KUKA KRL program: dai_chg_GRH_01.src, dai_chg_GRH_01.dat

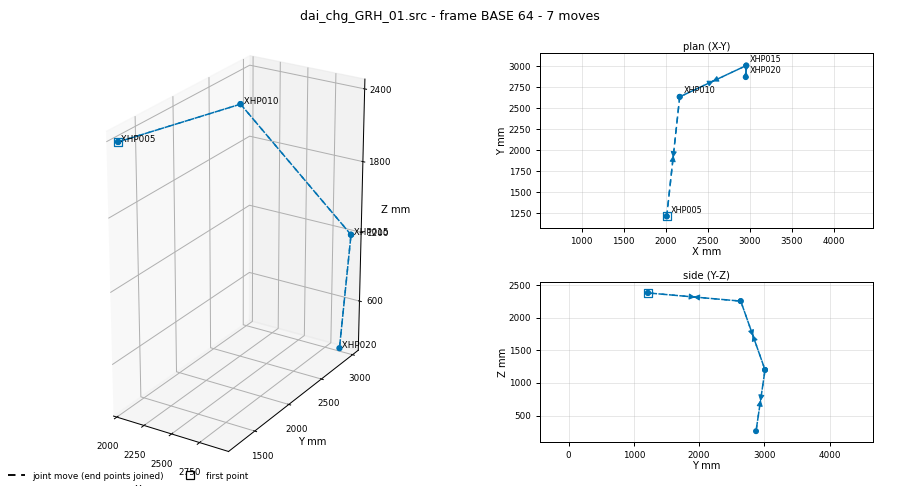
[picture p0: tool path of dai_chg_GRH_01.src in frame BASE 64, 7 of 9 moves have a stored position in this frame; points joined in program order, loops and branches not executed]
--- dai_chg_GRH_01.src ---
&ACCESS RVP
&REL 21
&COMMENT dai_chg_060GRH101
&USER PKL_AST
&PARAM version = 0.1
&PARAM DISKPATH = KRC:\R1\H_Prog
DEF dai_chg_GRH_01( )
;FOLD INI
  ;FOLD BASISTECH INI
    GLOBAL INTERRUPT DECL 3 WHEN $STOPMESS==TRUE DO IR_STOPM ( )
    BAS (#INITMOV,0 )
  ;ENDFOLD (BASISTECH INI)
;FOLD USER INI

;Make your modifications here
;FOLD COLLISION_V_3.01 INI ;%{E}
    IF (COLLISION_DATA[1].I_NR>0) THEN
    GLOBAL INTERRUPT DECL 21 WHEN $IN[COLLISION_DATA[1].I_NR]==FALSE DO COLLSTOP (1,0 )
    ENDIF
    IF (COLLISION_DATA[2].I_NR>0) THEN
    GLOBAL INTERRUPT DECL 22 WHEN $IN[COLLISION_DATA[2].I_NR]==FALSE DO COLLSTOP (2,0 )
    ENDIF
    IF (COLLISION_DATA[3].I_NR>0) THEN
    GLOBAL INTERRUPT DECL 23 WHEN $IN[COLLISION_DATA[3].I_NR]==FALSE DO COLLSTOP (3,0 )
    ENDIF
    IF (COLLISION_DATA[4].I_NR>0) THEN
    GLOBAL INTERRUPT DECL 24 WHEN $IN[COLLISION_DATA[4].I_NR]==FALSE DO COLLSTOP (4,0 )
    ENDIF
;ENDFOLD (Collision)

;ENDFOLD (USER INI)

;ENDFOLD (INI)
;FOLD ; Anlagenbezeichn: HC53_C    Stations-Nr: 060RB_100;%{PE}
;FOLD Parameters ;%{h}
;Params IlfProvider=kukaroboter.basistech.inlineforms.comments.comment; Kuka.Content=Anlagenbezeichn: HC53_C    Stations-Nr: 060RB_100
;ENDFOLD
;ENDFOLD
;FOLD ; Stand / Version: V1.0;%{PE}
;FOLD Parameters ;%{h}
;Params IlfProvider=kukaroboter.basistech.inlineforms.comments.comment; Kuka.Content=Stand / Version: V1.0
;ENDFOLD
;ENDFOLD
;FOLD ; Name Bearbeiter: EBZ-AE;%{PE}
;FOLD Parameters ;%{h}
;Params IlfProvider=kukaroboter.basistech.inlineforms.comments.comment; Kuka.Content=Name Bearbeiter: EBZ-AE
;ENDFOLD
;ENDFOLD
;FOLD ; Translator Version:29.01.2024 - Version 15.08;%{PE}
;FOLD Parameters ;%{h}
;Params IlfProvider=kukaroboter.basistech.inlineforms.comments.comment; Kuka.Content=Translator Version:29.01.2024 - Version 15.08
;ENDFOLD
;ENDFOLD


;FOLD ; This program has been cleaned by KANERT_Makro. High risk of crash!!! Check the program carefully before deleting this comment. ;%{PE}
;FOLD Parameters ;%{h}
;Params IlfProvider=kukaroboter.basistech.inlineforms.comments.comment; Kuka.Content=This program has been cleaned by KANERT_Makro. High risk of crash!!! Check the program carefully before deleting this comment.
;ENDFOLD
WAIT FOR FALSE
;ENDFOLD
REPEAT
;fold MSG_T1
MSG_SHOW("DAI_H_Prog",#quit,999,"dai_toolchange_0")
;endfold
; ***************************************
; A T T E N T I O N !!! Only drive in $T1
; A C H T U N G !!! Nur in $T1 abfahren
; ***************************************
UNTIL $T1 == TRUE
;FOLD PTP HOME Vel=100 % DEFAULT ;%{PE}
;FOLD Parameters ;%{h}
;Params IlfProvider=kukaroboter.basistech.inlineforms.movement.old; Kuka.IsGlobalPoint=False; Kuka.PointName=HOME; Kuka.BlendingEnabled=False; Kuka.MoveDataPtpName=DEFAULT; Kuka.VelocityPtp=100; Kuka.CurrentCDSetIndex=0; Kuka.MovementParameterFieldEnabled=True; IlfCommand=PTP
;ENDFOLD
$BWDSTART = FALSE
PDAT_ACT = PDEFAULT
FDAT_ACT = FHOME
BAS(#PTP_PARAMS, 100.0)
SET_CD_PARAMS (0)
PTP XHOME
;ENDFOLD

;Dynamische Pruefung Teil vorhanden
;FOLD PartPresent.CheckOff #1:5277, #2:5278, #3:1025, #4:1025, #5:1025, #6:1025, Bounce Time:100, Constant: Yes;%{PE}%
CheckPartPresent(5277,5278,1025,1025,1025,1025,100, True,FALSE)
;ENDFOLD
;FOLD DAI_GripValve.Valve2 State: Fixierstift Ausfahren Gs, Check: No, 060GRH101-QM1 ;%{PE}
ActuateValve(2,1, FALSE ,FALSE)
;ENDFOLD
;FOLD DAI_GripValve.Valve3 State: Spanner Oeffnen Gs, Check: No, 060GRH101-QM2 ;%{PE}
ActuateValve(3,1, FALSE ,FALSE)
;ENDFOLD
;FOLD DAI_GripValve.Valve4 State: Spanner Oeffnen Gs, Check: No, 060GRH101-QM3 ;%{PE}
ActuateValve(4,1, FALSE ,FALSE)
;ENDFOLD

;Greifer-Ventile betatigen/pruefen
;FOLD DAI_GripValveCheck.Valve2 State:Fixierstift Ausfahren Gs, 060GRH101-QM1;%{PE}%
CheckValveState(2,1)
;ENDFOLD
;FOLD DAI_GripValveCheck.Valve3 State:Spanner Oeffnen Gs, 060GRH101-QM2;%{PE}%
CheckValveState(3,1)
;ENDFOLD
;FOLD DAI_GripValveCheck.Valve4 State:Spanner Oeffnen Gs, 060GRH101-QM3;%{PE}%
CheckValveState(4,1)
;ENDFOLD

; Weg zu Ablageposition teachen
; Teach PTP-Way to depositing-position
;FOLD PTP HP005 Vel=100 % PDAT1 Tool[64]:Zero Base[64]:Zero ;%{PE}
;FOLD Parameters ;%{h}
;Params IlfProvider=kukaroboter.basistech.inlineforms.movement.old; Kuka.IsGlobalPoint=False; Kuka.PointName=HP005; Kuka.BlendingEnabled=False; Kuka.MoveDataPtpName=PDAT1; Kuka.VelocityPtp=100; Kuka.CurrentCDSetIndex=0; Kuka.MovementParameterFieldEnabled=True; IlfCommand=PTP
;ENDFOLD
$BWDSTART = FALSE
PDAT_ACT = PPDAT1
FDAT_ACT = FHP005
BAS(#PTP_PARAMS, 100.0)
SET_CD_PARAMS (0)
PTP XHP005
;ENDFOLD
;FOLD PTP HP010 Vel=100 % PDAT2 Tool[64]:Zero Base[64]:Zero ;%{PE}
;FOLD Parameters ;%{h}
;Params IlfProvider=kukaroboter.basistech.inlineforms.movement.old; Kuka.IsGlobalPoint=False; Kuka.PointName=HP010; Kuka.BlendingEnabled=False; Kuka.MoveDataPtpName=PDAT2; Kuka.VelocityPtp=100; Kuka.CurrentCDSetIndex=0; Kuka.MovementParameterFieldEnabled=True; IlfCommand=PTP
;ENDFOLD
$BWDSTART = FALSE
PDAT_ACT = PPDAT2
FDAT_ACT = FHP010
BAS(#PTP_PARAMS, 100.0)
SET_CD_PARAMS (0)
PTP XHP010
;ENDFOLD
;FOLD PTP HP015 Vel=100 % PDAT3 Tool[64]:Zero Base[64]:Zero ;%{PE}
;FOLD Parameters ;%{h}
;Params IlfProvider=kukaroboter.basistech.inlineforms.movement.old; Kuka.IsGlobalPoint=False; Kuka.PointName=HP015; Kuka.BlendingEnabled=False; Kuka.MoveDataPtpName=PDAT3; Kuka.VelocityPtp=100; Kuka.CurrentCDSetIndex=0; Kuka.MovementParameterFieldEnabled=True; IlfCommand=PTP
;ENDFOLD
$BWDSTART = FALSE
PDAT_ACT = PPDAT3
FDAT_ACT = FHP015
BAS(#PTP_PARAMS, 100.0)
SET_CD_PARAMS (0)
PTP XHP015
;ENDFOLD

; Ablageposition teachen
; depositing-position
;FOLD PTP HP020 Vel=100 % PDAT4 Tool[64]:Zero Base[64]:Zero ;%{PE}
;FOLD Parameters ;%{h}
;Params IlfProvider=kukaroboter.basistech.inlineforms.movement.old; Kuka.IsGlobalPoint=False; Kuka.PointName=HP020; Kuka.BlendingEnabled=False; Kuka.MoveDataPtpName=PDAT4; Kuka.VelocityPtp=100; Kuka.CurrentCDSetIndex=0; Kuka.MovementParameterFieldEnabled=True; IlfCommand=PTP
;ENDFOLD
$BWDSTART = FALSE
PDAT_ACT = PPDAT4
FDAT_ACT = FHP020
BAS(#PTP_PARAMS, 100.0)
SET_CD_PARAMS (0)
PTP XHP020
;ENDFOLD

;fold Ablageposition erreicht | depositing-position reeached
MSG_SHOW("DAI_H_Prog",#quit,999,"dai_toolchange_1")
;endfold
WAIT FOR  $IN[1026]==TRUE ;

REPEAT
;fold MSG_T1
MSG_SHOW("DAI_H_Prog",#quit,999,"dai_toolchange_0")
;endfold
; ***************************************
; A T T E N T I O N !!! Only drive in $T1
; A C H T U N G !!! Nur in $T1 abfahren
; ***************************************
UNTIL $T1 == TRUE

; Teache Weg zurueck zu Homeposition
; Teach PTP-way back to home
;FOLD PTP HP025 Vel=100 % PDAT5 Tool[64]:Zero Base[64]:Zero ;%{PE}
;FOLD Parameters ;%{h}
;Params IlfProvider=kukaroboter.basistech.inlineforms.movement.old; Kuka.IsGlobalPoint=False; Kuka.PointName=HP025; Kuka.BlendingEnabled=False; Kuka.MoveDataPtpName=PDAT5; Kuka.VelocityPtp=100; Kuka.CurrentCDSetIndex=0; Kuka.MovementParameterFieldEnabled=True; IlfCommand=PTP
;ENDFOLD
$BWDSTART = FALSE
PDAT_ACT = PPDAT5
FDAT_ACT = FHP025
BAS(#PTP_PARAMS, 100.0)
SET_CD_PARAMS (0)
PTP XHP025
;ENDFOLD
;FOLD PTP HP030 Vel=100 % PDAT6 Tool[64]:Zero Base[64]:Zero ;%{PE}
;FOLD Parameters ;%{h}
;Params IlfProvider=kukaroboter.basistech.inlineforms.movement.old; Kuka.IsGlobalPoint=False; Kuka.PointName=HP030; Kuka.BlendingEnabled=False; Kuka.MoveDataPtpName=PDAT6; Kuka.VelocityPtp=100; Kuka.CurrentCDSetIndex=0; Kuka.MovementParameterFieldEnabled=True; IlfCommand=PTP
;ENDFOLD
$BWDSTART = FALSE
PDAT_ACT = PPDAT6
FDAT_ACT = FHP030
BAS(#PTP_PARAMS, 100.0)
SET_CD_PARAMS (0)
PTP XHP030
;ENDFOLD
;FOLD PTP HP035 Vel=100 % PDAT7 Tool[64]:Zero Base[64]:Zero ;%{PE}
;FOLD Parameters ;%{h}
;Params IlfProvider=kukaroboter.basistech.inlineforms.movement.old; Kuka.IsGlobalPoint=False; Kuka.PointName=HP035; Kuka.BlendingEnabled=False; Kuka.MoveDataPtpName=PDAT7; Kuka.VelocityPtp=100; Kuka.CurrentCDSetIndex=0; Kuka.MovementParameterFieldEnabled=True; IlfCommand=PTP
;ENDFOLD
$BWDSTART = FALSE
PDAT_ACT = PPDAT7
FDAT_ACT = FHP035
BAS(#PTP_PARAMS, 100.0)
SET_CD_PARAMS (0)
PTP XHP035
;ENDFOLD

;FOLD PTP HOME Vel=100 % DEFAULT;%{PE}
;FOLD Parameters ;%{h}
;Params IlfProvider=kukaroboter.basistech.inlineforms.movement.old; Kuka.IsGlobalPoint=False; Kuka.PointName=HOME; Kuka.BlendingEnabled=False; Kuka.MoveDataPtpName=DEFAULT; Kuka.VelocityPtp=100; Kuka.CurrentCDSetIndex=0; Kuka.MovementParameterFieldEnabled=True; IlfCommand=PTP
;ENDFOLD
$BWDSTART = FALSE
PDAT_ACT = PDEFAULT
FDAT_ACT = FHOME
BAS(#PTP_PARAMS, 100.0)
SET_CD_PARAMS (0)
PTP XHOME
;ENDFOLD

END

--- dai_chg_GRH_01.dat ---
&ACCESS RVP
&REL 22
&COMMENT dai_chg_060GRH101
&USER PKL_AST
&PARAM version = 0.1
&PARAM DISKPATH = KRC:\R1\H_Prog
DEFDAT  DAI_CHG_GRH_01
;FOLD EXTERNAL DECLARATIONS;%{PE}%MKUKATPBASIS,%CEXT,%VCOMMON,%P
;FOLD BASISTECH EXT;%{PE}%MKUKATPBASIS,%CEXT,%VEXT,%P
EXT  BAS (BAS_COMMAND  :IN,REAL  :IN )
DECL INT SUCCESS
;ENDFOLD (BASISTECH EXT)
;FOLD USER EXT;%{E}%MKUKATPUSER,%CEXT,%VEXT,%P
;Make here your modifications
;FOLD COLLISION
EXT  COLLSTOP (INT  :IN,INT  :IN )
;ENDFOLD  (Collision)
;ENDFOLD (USER EXT)
;ENDFOLD (EXTERNAL DECLERATIONS)
DECL INT handle,answer
DECL BASIS_SUGG_T LAST_BASIS={POINT1[] "P0                      ",POINT2[] "P0                      ",CP_PARAMS[] "CPDAT0                  ",PTP_PARAMS[] "PDAT0                   ",CONT[] "                        ",CP_VEL[] "2                       ",PTP_VEL[] "100                     ",SYNC_PARAMS[] "SYNCDAT                 ",SPL_NAME[] "S0                      "}
DECL MODULEPARAM_T LAST_TP_PARAMS={PARAMS[] "Kuka.PointName=HP025; Kuka.FrameData.base_no=64; Kuka.FrameData.tool_no=64; Kuka.FrameData.ipo_frame=#BASE; Kuka.FrameData.point2=; Kuka.isglobalpoint=False; Kuka.MoveDataPtpName=PDAT5; Kuka.MovementDataPdat.apo_mode=#CDIS; Kuka.MovementDataPdat.apo_dist=100; Kuka.MovementData.acc=100; Kuka.MovementData.gear_jerk=100; Kuka.MovementData.exax_ign=0; Kuka.VelocityPtp=100; Kuka.BlendingEnabled=False; Kuka.CurrentCDSetIndex=0; Kuka.MovementData.vel=100; Kuka.APXEnabled=False; Kuka.Content=Anlagenbezeichn: VU52_A    Stations-Nr: 030RB_100; DAI_GRIPVALVECHECK.LSTSTATES2=1; DAI_GRIPVALVECHECK.FREEVALVETEXT2=060GRH101-QM1; DAI_GRIPVALVE.LSTSTATES2=1; DAI_GRIPVALVE.LSTCHECK=FALSE; DAI_GRIPVALVE.FREEVALVETEXT2=060GRH101-QM1; DAI_GRIPVALVE.LSTSTATES3=1; DAI_GRIPVALVE.FREEVALVETEXT3=060GRH101-QM2; DAI_GRIPVALVE.LSTSTATES4=1; DAI_GRIPVALVE.FREEVALVETEXT4=060GRH101-QM3"}

; E6POS Declarations
DECL E6POS XHP005={X 2014.02515,Y 1215.68958,Z 2380.21460,A -29.0518417,B -0.0196952634,C -149.520157,S 18,T 11,E1 -1339.73975,E2 0.0,E3 0.0,E4 0.0,E5 0.0,E6 0.0}
DECL E6POS XHP010={X 2168.62500,Y 2638.36572,Z 2254.92554,A 83.5215454,B 55.9669724,C 6.17859936,S 22,T 27,E1 -1642.06177,E2 0.0,E3 0.0,E4 0.0,E5 0.0,E6 0.0}
DECL E6POS XHP015={X 2960.82275,Y 3010.84717,Z 1200.10413,A 87.7378616,B 73.0204544,C 10.8167992,S 22,T 27,E1 -2360.99463,E2 0.0,E3 0.0,E4 0.0,E5 0.0,E6 0.0}
DECL E6POS XHP020={X 2954.79980,Y 2872.63354,Z 260.112061,A -110.254951,B 89.8050232,C 171.444794,S 22,T 57,E1 -2360.99463,E2 0.0,E3 0.0,E4 0.0,E5 0.0,E6 0.0}
DECL E6POS XHP025={X 2960.82275,Y 3010.84717,Z 1200.10413,A 87.7378616,B 73.0204544,C 10.8167992,S 22,T 27,E1 -2360.99463,E2 0.0,E3 0.0,E4 0.0,E5 0.0,E6 0.0}
DECL E6POS XHP030={X 2168.62500,Y 2638.36572,Z 2254.92554,A 83.5215454,B 55.9669724,C 6.17859936,S 22,T 27,E1 -1642.06177,E2 0.0,E3 0.0,E4 0.0,E5 0.0,E6 0.0}
DECL E6POS XHP035={X 2014.02515,Y 1215.68958,Z 2380.21460,A -29.0518417,B -0.0196952634,C -149.520157,S 18,T 11,E1 -1339.73975,E2 0.0,E3 0.0,E4 0.0,E5 0.0,E6 0.0}

; PDAT/LDAT Declarations
DECL PDAT PPDAT1={VEL 100.000,ACC 100.000,APO_DIST 100.000,APO_MODE #CDIS,GEAR_JERK 100.000,EXAX_IGN 0}
DECL PDAT PPDAT2={VEL 100.000,ACC 100.000,APO_DIST 100.000,APO_MODE #CDIS,GEAR_JERK 100.000,EXAX_IGN 0}
DECL PDAT PPDAT3={VEL 100.000,ACC 100.000,APO_DIST 100.000,APO_MODE #CDIS,GEAR_JERK 100.000,EXAX_IGN 0}
DECL PDAT PPDAT4={VEL 100.000,ACC 100.000,APO_DIST 100.000,APO_MODE #CDIS,GEAR_JERK 100.000,EXAX_IGN 0}
DECL PDAT PPDAT5={VEL 100.000,ACC 100.000,APO_DIST 100.000,APO_MODE #CDIS,GEAR_JERK 100.000,EXAX_IGN 0}
DECL PDAT PPDAT6={VEL 100.000,ACC 100.000,APO_DIST 100.000,APO_MODE #CDIS,GEAR_JERK 100.000,EXAX_IGN 0}
DECL PDAT PPDAT7={VEL 100.000,ACC 100.000,APO_DIST 100.000,APO_MODE #CDIS,GEAR_JERK 100.000,EXAX_IGN 0}

; FDAT Declarations
DECL FDAT FHOME={TOOL_NO 0,BASE_NO 0,IPO_FRAME #BASE,POINT2[] " "}
DECL FDAT FHP005={TOOL_NO 64,BASE_NO 64,IPO_FRAME #BASE,POINT2[] " "}
DECL FDAT FHP010={TOOL_NO 64,BASE_NO 64,IPO_FRAME #BASE,POINT2[] " "}
DECL FDAT FHP015={TOOL_NO 64,BASE_NO 64,IPO_FRAME #BASE,POINT2[] " "}
DECL FDAT FHP020={TOOL_NO 64,BASE_NO 64,IPO_FRAME #BASE,POINT2[] " "}
DECL FDAT FHP025={TOOL_NO 64,BASE_NO 64,IPO_FRAME #BASE,POINT2[] " "}
DECL FDAT FHP030={TOOL_NO 64,BASE_NO 64,IPO_FRAME #BASE,POINT2[] " "}
DECL FDAT FHP035={TOOL_NO 64,BASE_NO 64,IPO_FRAME #BASE,POINT2[] " "}

ENDDAT
